(* Logix 5000 project; controller Ejercicio_Numero_5 Emulate 5570 rev 33.11; software revision 33.00 *)

TASK T00_MainTask (continuous, watchdog 500 ms) : P00_MainProgram

MODULES
   Local : Emulate 5570 (ICP 3, rev 33.11)
END_MODULES

PROGRAM P00_MainProgram   (* main routine R00_MainRoutine *)
VAR
   AT_ENTRY_1 : BOOL := 1;
   AT_ENTRY_2 : BOOL := 1;
   AT_EXIT : BOOL := 1;
   AT_TRANSFER_1 : BOOL;
   AT_TRANSFER_2 : BOOL;
   AUTOMATICO : BOOL := 1;
   BOX_LEAVING_1 : BOOL := 1;
   CONVEYOR_1 : BOOL;
   CONVEYOR_1_HMI : BOOL;
   CONVEYOR_2 : BOOL;
   CONVEYOR_2_HMI : BOOL;
   CONVEYOR_LEFT : BOOL;
   CONVEYOR_LEFT_1 : BOOL;
   CONVEYOR_RIGHT : BOOL;
   CONVEYOR_RIGHT_1 : BOOL;
   EXIT_CONVEYOR : BOOL := 1;
   EXIT_CONVEYOR_HMI : BOOL;
   LOAD_1 : BOOL;
   LOAD_1_HMI : BOOL;
   LOAD_2 : BOOL;
   LOAD_2_HMI : BOOL;
   LOADING_1 : BOOL;
   LOADING_2 : BOOL;
   MANUAL : BOOL;
   MOVING_LEFT_1 : BOOL;
   MOVING_LEFT_2 : BOOL;
   OSF : BOOL;
   RESET : BOOL;
   SEQUENCER_LEFT : DINT;
   SEQUENCER_RIGHT : DINT;
   SHOT_1 : BOOL;
   SHOT_2 : BOOL;
   START : BOOL;
   START_CYCLE : BOOL := 1;
   STOP : BOOL := 1;
   STOP_CONVEYOR_LEFT : BOOL;
   STORAGE_BIT : BOOL := 1;
   TIMER : TIMER[10] := ([0].PRE := 4000, [1].PRE := 6500, [1].ACC := 6500, [2].PRE := 3300, [2].EN := 1, [2].DN := 1);
   TRANSFER : BOOL;
   TRANSFER_LEFT_1 : BOOL;
   TRANSFER_LEFT_1_HMI : BOOL;
   TRANSFER_LEFT_2 : BOOL;
   TRANSFER_LEFT_2_HMI : BOOL;
END_VAR

ROUTINE R00_MainRoutine   (* ladder *)
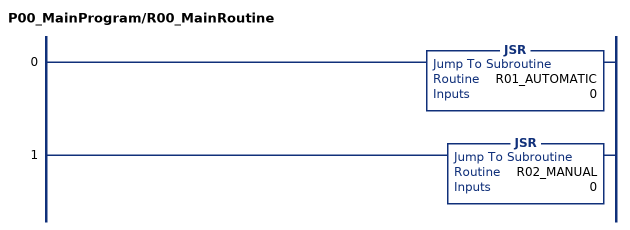
   0: JSR(R01_AUTOMATIC,0);
   1: JSR(R02_MANUAL,0);
END_ROUTINE

ROUTINE R01_AUTOMATIC   (* ladder *)
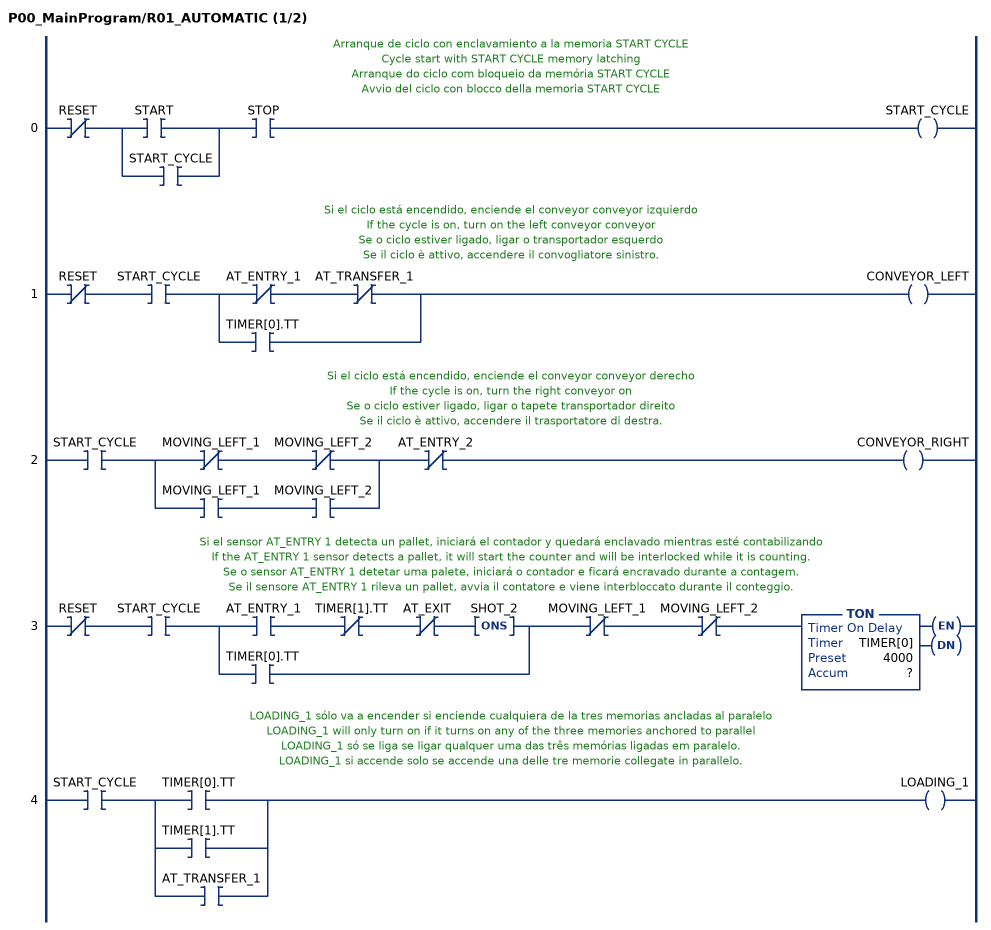
   // Arranque de ciclo con enclavamiento a la memoria START CYCLE
   // Cycle start with START CYCLE memory latching
   // Arranque do ciclo com bloqueio da memória START CYCLE
   // Avvio del ciclo con blocco della memoria START CYCLE
   0: XIO(RESET)[XIC(START) ,XIC(START_CYCLE) ]XIC(STOP)OTE(START_CYCLE);
   // Si el ciclo está encendido, enciende el conveyor conveyor izquierdo
   // If the cycle is on, turn on the left conveyor conveyor
   // Se o ciclo estiver ligado, ligar o transportador esquerdo
   // Se il ciclo è attivo, accendere il convogliatore sinistro.
   1: XIO(RESET)XIC(START_CYCLE)[XIO(AT_ENTRY_1) XIO(AT_TRANSFER_1) ,XIC(TIMER[0].TT) ]OTE(CONVEYOR_LEFT);
   // Si el ciclo está encendido, enciende el conveyor conveyor derecho
   // If the cycle is on, turn the right conveyor on
   // Se o ciclo estiver ligado, ligar o tapete transportador direito
   // Se il ciclo è attivo, accendere il trasportatore di destra.
   2: XIC(START_CYCLE)[XIO(MOVING_LEFT_1) XIO(MOVING_LEFT_2) ,XIC(MOVING_LEFT_1) XIC(MOVING_LEFT_2) ]XIO(AT_ENTRY_2)OTE(CONVEYOR_RIGHT);
   // Si el sensor AT_ENTRY 1 detecta un pallet, iniciará el contador y quedará enclavado mientras esté contabilizando
   // If the AT_ENTRY 1 sensor detects a pallet, it will start the counter and will be interlocked while it is counting.
   // Se o sensor AT_ENTRY 1 detetar uma palete, iniciará o contador e ficará encravado durante a contagem.
   // Se il sensore AT_ENTRY 1 rileva un pallet, avvia il contatore e viene interbloccato durante il conteggio.
   3: XIO(RESET)XIC(START_CYCLE)[XIC(AT_ENTRY_1) XIO(TIMER[1].TT) XIO(AT_EXIT) ONS(SHOT_2) ,XIC(TIMER[0].TT) ]XIO(MOVING_LEFT_1)XIO(MOVING_LEFT_2)TON(TIMER[0],?,?);
   // LOADING_1 sólo va a encender si enciende cualquiera de la tres memorias ancladas al paralelo
   // LOADING_1 will only turn on if it turns on any of the three memories anchored to parallel
   // LOADING_1 só se liga se ligar qualquer uma das três memórias ligadas em paralelo.
   // LOADING_1 si accende solo se accende una delle tre memorie collegate in parallelo.
   4: XIC(START_CYCLE)[XIC(TIMER[0].TT) ,XIC(TIMER[1].TT) ,XIC(AT_TRANSFER_1) ]OTE(LOADING_1);
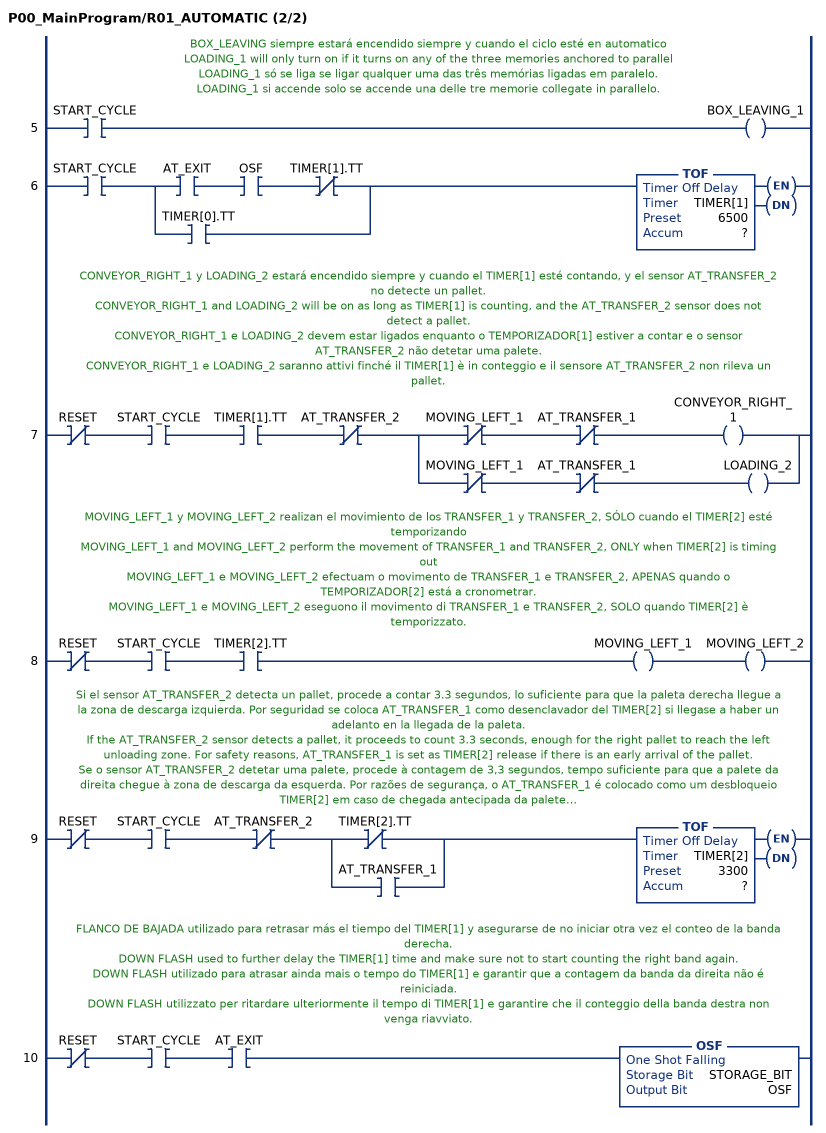
   // BOX_LEAVING siempre estará encendido siempre y cuando el ciclo esté en automatico
   // LOADING_1 will only turn on if it turns on any of the three memories anchored to parallel
   // LOADING_1 só se liga se ligar qualquer uma das três memórias ligadas em paralelo.
   // LOADING_1 si accende solo se accende una delle tre memorie collegate in parallelo.
   5: XIC(START_CYCLE)OTE(BOX_LEAVING_1);
   6: XIC(START_CYCLE)[XIC(AT_EXIT) XIC(OSF) XIO(TIMER[1].TT) ,XIC(TIMER[0].TT) ]TOF(TIMER[1],?,?);
   // CONVEYOR_RIGHT_1 y LOADING_2 estará encendido siempre y cuando el TIMER[1] esté contando, y el sensor AT_TRANSFER_2 no detecte un pallet.
   // CONVEYOR_RIGHT_1 and LOADING_2 will be on as long as TIMER[1] is counting, and the AT_TRANSFER_2 sensor does not detect a pallet.
   // CONVEYOR_RIGHT_1 e LOADING_2 devem estar ligados enquanto o TEMPORIZADOR[1] estiver a contar e o sensor AT_TRANSFER_2 não detetar uma palete.
   // CONVEYOR_RIGHT_1 e LOADING_2 saranno attivi finché il TIMER[1] è in conteggio e il sensore AT_TRANSFER_2 non rileva un pallet.
   7: XIO(RESET)XIC(START_CYCLE)XIC(TIMER[1].TT)XIO(AT_TRANSFER_2)[XIO(MOVING_LEFT_1) XIO(AT_TRANSFER_1) OTE(CONVEYOR_RIGHT_1) ,XIO(MOVING_LEFT_1) XIO(AT_TRANSFER_1) OTE(LOADING_2) ];
   // MOVING_LEFT_1 y MOVING_LEFT_2 realizan el movimiento de los TRANSFER_1 y TRANSFER_2, SÓLO cuando el TIMER[2] esté temporizando
   // MOVING_LEFT_1 and MOVING_LEFT_2 perform the movement of TRANSFER_1 and TRANSFER_2, ONLY when TIMER[2] is timing out
   // MOVING_LEFT_1 e MOVING_LEFT_2 efectuam o movimento de TRANSFER_1 e TRANSFER_2, APENAS quando o TEMPORIZADOR[2] está a cronometrar.
   // MOVING_LEFT_1 e MOVING_LEFT_2 eseguono il movimento di TRANSFER_1 e TRANSFER_2, SOLO quando TIMER[2] è temporizzato.
   8: XIO(RESET)XIC(START_CYCLE)XIC(TIMER[2].TT)OTE(MOVING_LEFT_1)OTE(MOVING_LEFT_2);
   // Si el sensor AT_TRANSFER_2 detecta un pallet, procede a contar 3.3 segundos, lo suficiente para que la paleta derecha llegue a la zona de descarga izquierda. Por seguridad se coloca AT_TRANSFER_1 como desenclavador del TIMER[2] si llegase a haber un adelanto en la llegada de la paleta.
   // If the AT_TRANSFER_2 sensor detects a pallet, it proceeds to count 3.3 seconds, enough for the right pallet to reach the left unloading zone. For safety reasons, AT_TRANSFER_1 is set as TIMER[2] release if there is an early arrival of the pallet.
   // Se o sensor AT_TRANSFER_2 detetar uma palete, procede à contagem de 3,3 segundos, tempo suficiente para que a palete da direita chegue à zona de descarga da esquerda. Por razões de segurança, o AT_TRANSFER_1 é colocado como um desbloqueio TIMER[2] em caso de chegada antecipada da palete.
   // Se il sensore AT_TRANSFER_2 rileva un pallet, procede al conteggio di 3,3 secondi, tempo sufficiente affinché il pallet destro raggiunga la zona di scarico sinistra. Per motivi di sicurezza, AT_TRANSFER_1 viene posizionato come rilascio TIMER[2] in caso di arrivo anticipato del pallet.
   9: XIO(RESET)XIC(START_CYCLE)XIO(AT_TRANSFER_2)[XIO(TIMER[2].TT) ,XIC(AT_TRANSFER_1) ]TOF(TIMER[2],?,?);
   // FLANCO DE BAJADA utilizado para retrasar más el tiempo del TIMER[1] y asegurarse de no iniciar otra vez el conteo de la banda derecha.
   // DOWN FLASH used to further delay the TIMER[1] time and make sure not to start counting the right band again.
   // DOWN FLASH utilizado para atrasar ainda mais o tempo do TIMER[1] e garantir que a contagem da banda da direita não é reiniciada.
   // DOWN FLASH utilizzato per ritardare ulteriormente il tempo di TIMER[1] e garantire che il conteggio della banda destra non venga riavviato.
   10: XIO(RESET)XIC(START_CYCLE)XIC(AT_EXIT)OSF(STORAGE_BIT,OSF);
END_ROUTINE

ROUTINE R02_MANUAL   (* ladder *)
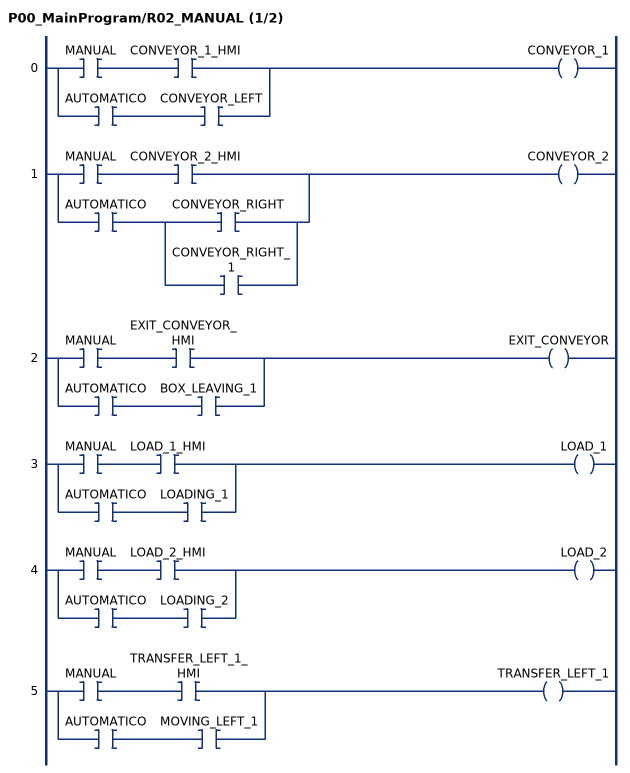
   0: [XIC(MANUAL) XIC(CONVEYOR_1_HMI) ,XIC(AUTOMATICO) XIC(CONVEYOR_LEFT) ]OTE(CONVEYOR_1);
   1: [XIC(MANUAL) XIC(CONVEYOR_2_HMI) ,XIC(AUTOMATICO) [XIC(CONVEYOR_RIGHT) ,XIC(CONVEYOR_RIGHT_1) ] ]OTE(CONVEYOR_2);
   2: [XIC(MANUAL) XIC(EXIT_CONVEYOR_HMI) ,XIC(AUTOMATICO) XIC(BOX_LEAVING_1) ]OTE(EXIT_CONVEYOR);
   3: [XIC(MANUAL) XIC(LOAD_1_HMI) ,XIC(AUTOMATICO) XIC(LOADING_1) ]OTE(LOAD_1);
   4: [XIC(MANUAL) XIC(LOAD_2_HMI) ,XIC(AUTOMATICO) XIC(LOADING_2) ]OTE(LOAD_2);
   5: [XIC(MANUAL) XIC(TRANSFER_LEFT_1_HMI) ,XIC(AUTOMATICO) XIC(MOVING_LEFT_1) ]OTE(TRANSFER_LEFT_1);
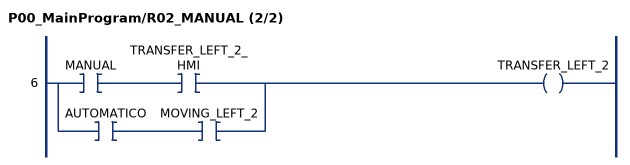
   6: [XIC(MANUAL) XIC(TRANSFER_LEFT_2_HMI) ,XIC(AUTOMATICO) XIC(MOVING_LEFT_2) ]OTE(TRANSFER_LEFT_2);
END_ROUTINE
END_PROGRAM
